{attribute addProperty BoxType "EK1122-0000-0018"}
{attribute addProperty Id "Beckhoff_EPP6xxxsub_EK1100EK1100_179A0949162A_0001_EPP6001_0002_0016EPP6001_7904467646658.25A_0002_EPP6001_0002_0017EPP6001_7904467646658.25A_0003_EPP6001_0002_0018EPP6001_7904467646658.25A_0004_EPP6002_0002_0016EPP6002_320F021A850106.25A_0005_EPP6002_0002_0017EPP6002_320F021A850106.25A_0006_EPP6002_0002_0018EPP6002_FC20A988850106.25A_0007_EPP6002_0002_0019EPP6002_FC20A988850106.25A_0008_EPP6090_0000_0017EPP6090_7D66C95013016.25A_0009_EPP6228_0022_0016EPP6228_E048681B27434.25"}
{attribute addProperty CRC "1476671912"}
{attribute addProperty SizeInBites "5218"}
{attribute addProperty SizeInBytes "652.25"}
TYPE Beckhoff_EPP6xxxEK1122_580439A8 EXTENDS EK1122_179A0949 :
STRUCT
	{attribute addProperty Name "Beckhoff_EPP6xxxsub_EK1100"}
	Beckhoff_EPP6xxxsub_EK1100 : EK1100_179A0949;
	{attribute addProperty Name "A_0001_EPP6001_0002_0016"}
	A_0001_EPP6001_0002_0016 : EPP6001_79044676;
	{attribute addProperty Name "A_0002_EPP6001_0002_0017"}
	A_0002_EPP6001_0002_0017 : EPP6001_79044676;
	{attribute addProperty Name "A_0003_EPP6001_0002_0018"}
	A_0003_EPP6001_0002_0018 : EPP6001_79044676;
	{attribute addProperty Name "A_0004_EPP6002_0002_0016"}
	A_0004_EPP6002_0002_0016 : EPP6002_320F021A;
	{attribute addProperty Name "A_0005_EPP6002_0002_0017"}
	A_0005_EPP6002_0002_0017 : EPP6002_320F021A;
	{attribute addProperty Name "A_0006_EPP6002_0002_0018"}
	A_0006_EPP6002_0002_0018 : EPP6002_FC20A988;
	{attribute addProperty Name "A_0007_EPP6002_0002_0019"}
	A_0007_EPP6002_0002_0019 : EPP6002_FC20A988;
	{attribute addProperty Name "A_0008_EPP6090_0000_0017"}
	A_0008_EPP6090_0000_0017 : EPP6090_7D66C950;
	{attribute addProperty Name "A_0009_EPP6228_0022_0016"}
	A_0009_EPP6228_0022_0016 : EPP6228_E048681B;
END_STRUCT
END_TYPE

(* stored: Version 1.2.0.0, ProductVersion 3.1.4024.9
   DUT Beckhoff_EPP6xxxEK1122_580439A8: Id {c7a2e2e7-31b6-4360-8b78-10278d1cba77} *)
